    UF : 0, UT : 6,      CONFIG : 'N U T, 0, 0, 0',
    X =  237.679  mm,    Y =   97.904  mm,    Z =   677.007  mm,
    W =  -181.004 deg,    P =   0.018 deg,    R =   -1.000 deg
};
P[413]{
   GP1:
    UF : 0, UT : 6,      CONFIG : 'N U T, 0, 0, 0',
    X =  239.805  mm,    Y =   100.038  mm,    Z =   678.567  mm,
    W =  -180.980 deg,    P =   0.017 deg,    R =   -1.000 deg
};
P[414]{
   GP1:
    UF : 0, UT : 6,      CONFIG : 'N U T, 0, 0, 0',
    X =  237.603  mm,    Y =   102.637  mm,    Z =   678.250  mm,
    W =  -180.939 deg,    P =   0.016 deg,    R =   -1.000 deg
};
P[415]{
   GP1:
    UF : 0, UT : 6,      CONFIG : 'N U T, 0, 0, 0',
    X =  237.914  mm,    Y =   109.032  mm,    Z =   679.196  mm,
    W =  -180.916 deg,    P =   0.016 deg,    R =   -1.000 deg
};
P[416]{
   GP1:
    UF : 0, UT : 6,      CONFIG : 'N U T, 0, 0, 0',
    X =  238.466  mm,    Y =   114.556  mm,    Z =   679.491  mm,
    W =  -180.917 deg,    P =   0.016 deg,    R =   -1.000 deg
};
P[417]{
   GP1:
    UF : 0, UT : 6,      CONFIG : 'N U T, 0, 0, 0',
    X =  237.988  mm,    Y =   117.959  mm,    Z =   679.696  mm,
    W =  -180.951 deg,    P =   0.017 deg,    R =   -1.000 deg
};
P[418]{
   GP1:
    UF : 0, UT : 6,      CONFIG : 'N U T, 0, 0, 0',
    X =  237.933  mm,    Y =   124.350  mm,    Z =   679.696  mm,
    W =  -180.999 deg,    P =   0.017 deg,    R =   -1.000 deg
};
P[419]{
   GP1:
    UF : 0, UT : 6,      CONFIG : 'N U T, 0, 0, 0',
    X =  238.236  mm,    Y =   206.397  mm,    Z =   679.696  mm,
    W =  -180.000 deg,    P =   0.000 deg,    R =   0.000 deg
};
P[420]{
   GP1:
    UF : 0, UT : 6,      CONFIG : 'N U T, 0, 0, 0',
    X =  201.883  mm,    Y =   206.397  mm,    Z =   677.551  mm,
    W =  -180.000 deg,    P =   0.000 deg,    R =   0.000 deg
};
P[421]{
   GP1:
    UF : 0, UT : 6,      CONFIG : 'N U T, 0, 0, 0',
    X =  202.738  mm,    Y =   124.967  mm,    Z =   677.551  mm,
    W =  -181.191 deg,    P =   0.021 deg,    R =   -1.000 deg
};
P[422]{
   GP1:
    UF : 0, UT : 6,      CONFIG : 'N U T, 0, 0, 0',
    X =  202.486  mm,    Y =   119.434  mm,    Z =   677.551  mm,
    W =  -181.103 deg,    P =   0.019 deg,    R =   -1.000 deg
};
P[423]{
   GP1:
    UF : 0, UT : 6,      CONFIG : 'N U T, 0, 0, 0',
    X =  203.228  mm,    Y =   114.890  mm,    Z =   677.970  mm,
    W =  -180.965 deg,    P =   0.017 deg,    R =   -1.000 deg
};
P[424]{
   GP1:
    UF : 0, UT : 6,      CONFIG : 'N U T, 0, 0, 0',
    X =  202.797  mm,    Y =   108.893  mm,    Z =   678.745  mm,
    W =  -180.839 deg,    P =   0.015 deg,    R =   -1.000 deg
};
P[425]{
   GP1:
    UF : 0, UT : 6,      CONFIG : 'N U T, 0, 0, 0',
    X =  202.869  mm,    Y =   103.650  mm,    Z =   678.789  mm,
    W =  -180.846 deg,    P =   0.015 deg,    R =   -1.000 deg
};
P[426]{
   GP1:
    UF : 0, UT : 6,      CONFIG : 'N U T, 0, 0, 0',
    X =  202.572  mm,    Y =   100.291  mm,    Z =   678.701  mm,
    W =  -180.857 deg,    P =   0.015 deg,    R =   -1.000 deg
};
P[427]{
   GP1:
    UF : 0, UT : 6,      CONFIG : 'N U T, 0, 0, 0',
    X =  202.760  mm,    Y =   96.899  mm,    Z =   677.464  mm,
    W =  -180.877 deg,    P =   0.015 deg,    R =   -1.000 deg
};
P[428]{
   GP1:
    UF : 0, UT : 6,      CONFIG : 'N U T, 0, 0, 0',
    X =  203.006  mm,    Y =   91.575  mm,    Z =   677.087  mm,
    W =  -180.968 deg,    P =   0.017 deg,    R =   -1.000 deg
};
P[429]{
   GP1:
    UF : 0, UT : 6,      CONFIG : 'N U T, 0, 0, 0',
    X =  202.936  mm,    Y =   85.805  mm,    Z =   677.228  mm,
    W =  -181.086 deg,    P =   0.019 deg,    R =   -1.000 deg
};
P[430]{
   GP1:
    UF : 0, UT : 6,      CONFIG : 'N U T, 0, 0, 0',
    X =  202.752  mm,    Y =   80.302  mm,    Z =   677.133  mm,
    W =  -181.183 deg,    P =   0.021 deg,    R =   -1.000 deg
};
P[431]{
   GP1:
    UF : 0, UT : 6,      CONFIG : 'N U T, 0, 0, 0',
    X =  203.266  mm,    Y =   74.595  mm,    Z =   677.308  mm,
    W =  -181.243 deg,    P =   0.022 deg,    R =   -1.000 deg
};
P[432]{
   GP1:
    UF : 0, UT : 6,      CONFIG : 'N U T, 0, 0, 0',
    X =  202.857  mm,    Y =   69.136  mm,    Z =   677.567  mm,
    W =  -181.285 deg,    P =   0.022 deg,    R =   -1.000 deg
};
P[433]{
   GP1:
    UF : 0, UT : 6,      CONFIG : 'N U T, 0, 0, 0',
    X =  202.244  mm,    Y =   64.466  mm,    Z =   677.604  mm,
    W =  -181.312 deg,    P =   0.023 deg,    R =   -1.000 deg
};
P[434]{
   GP1:
    UF : 0, UT : 6,      CONFIG : 'N U T, 0, 0, 0',
    X =  202.914  mm,    Y =   58.122  mm,    Z =   677.421  mm,
    W =  -181.367 deg,    P =   0.024 deg,    R =   -1.000 deg
};
P[435]{
   GP1:
    UF : 0, UT : 6,      CONFIG : 'N U T, 0, 0, 0',
    X =  203.053  mm,    Y =   53.855  mm,    Z =   677.512  mm,
    W =  -181.395 deg,    P =   0.024 deg,    R =   -1.000 deg
};
P[436]{
   GP1:
    UF : 0, UT : 6,      CONFIG : 'N U T, 0, 0, 0',
    X =  202.843  mm,    Y =   46.563  mm,    Z =   675.931  mm,
    W =  -181.419 deg,    P =   0.025 deg,    R =   -1.000 deg
};
P[437]{
   GP1:
    UF : 0, UT : 6,      CONFIG : 'N U T, 0, 0, 0',
    X =  203.318  mm,    Y =   42.100  mm,    Z =   674.942  mm,
    W =  -181.434 deg,    P =   0.025 deg,    R =   -1.000 deg
};
P[438]{
   GP1:
    UF : 0, UT : 6,      CONFIG : 'N U T, 0, 0, 0',
    X =  202.881  mm,    Y =   39.256  mm,    Z =   674.563  mm,
    W =  -181.438 deg,    P =   0.025 deg,    R =   -1.000 deg
};
P[439]{
   GP1:
    UF : 0, UT : 6,      CONFIG : 'N U T, 0, 0, 0',
    X =  203.131  mm,    Y =   34.198  mm,    Z =   674.988  mm,
    W =  -181.441 deg,    P =   0.025 deg,    R =   -1.000 deg
};
P[440]{
   GP1:
    UF : 0, UT : 6,      CONFIG : 'N U T, 0, 0, 0',
    X =  202.832  mm,    Y =   28.738  mm,    Z =   675.954  mm,
    W =  -181.416 deg,    P =   0.025 deg,    R =   -1.000 deg
};
P[441]{
   GP1:
    UF : 0, UT : 6,      CONFIG : 'N U T, 0, 0, 0',
    X =  202.744  mm,    Y =   23.472  mm,    Z =   676.873  mm,
    W =  -181.376 deg,    P =   0.024 deg,    R =   -1.000 deg
};
P[442]{
   GP1:
    UF : 0, UT : 6,      CONFIG : 'N U T, 0, 0, 0',
    X =  202.866  mm,    Y =   17.338  mm,    Z =   677.956  mm,
    W =  -181.263 deg,    P =   0.022 deg,    R =   -1.000 deg
};
P[443]{
   GP1:
    UF : 0, UT : 6,      CONFIG : 'N U T, 0, 0, 0',
    X =  203.265  mm,    Y =   12.113  mm,    Z =   677.623  mm,
    W =  -181.138 deg,    P =   0.020 deg,    R =   -1.000 deg
};
P[444]{
   GP1:
    UF : 0, UT : 6,      CONFIG : 'N U T, 0, 0, 0',
    X =  202.579  mm,    Y =   6.550  mm,    Z =   676.710  mm,
    W =  -180.997 deg,    P =   0.017 deg,    R =   -1.000 deg
};
P[445]{
   GP1:
    UF : 0, UT : 6,      CONFIG : 'N U T, 0, 0, 0',
    X =  202.981  mm,    Y =   2.035  mm,    Z =   675.441  mm,
    W =  -180.903 deg,    P =   0.016 deg,    R =   -1.000 deg
};
P[446]{
   GP1:
    UF : 0, UT : 6,      CONFIG : 'N U T, 0, 0, 0',
    X =  201.883  mm,    Y =   -0.623  mm,    Z =   676.010  mm,
    W =  -180.856 deg,    P =   0.015 deg,    R =   -1.000 deg
};
P[447]{
   GP1:
    UF : 0, UT : 6,      CONFIG : 'N U T, 0, 0, 0',
    X =  202.866  mm,    Y =   -4.118  mm,    Z =   675.410  mm,
    W =  -180.726 deg,    P =   0.013 deg,    R =   -1.000 deg
};
P[448]{
   GP1:
    UF : 0, UT : 6,      CONFIG : 'N U T, 0, 0, 0',
    X =  202.877  mm,    Y =   -10.672  mm,    Z =   675.669  mm,
    W =  -180.524 deg,    P =   0.009 deg,    R =   -1.000 deg
};
P[449]{
   GP1:
    UF : 0, UT : 6,      CONFIG : 'N U T, 0, 0, 0',
    X =  202.997  mm,    Y =   -15.857  mm,    Z =   675.460  mm,
    W =  -180.390 deg,    P =   0.007 deg,    R =   -1.000 deg
};
P[450]{
   GP1:
    UF : 0, UT : 6,      CONFIG : 'N U T, 0, 0, 0',
    X =  202.823  mm,    Y =   -21.947  mm,    Z =   675.573  mm,
    W =  -180.109 deg,    P =   0.002 deg,    R =   -0.999 deg
};
P[451]{
   GP1:
    UF : 0, UT : 6,      CONFIG : 'N U T, 0, 0, 0',
    X =  203.057  mm,    Y =   -65.498  mm,    Z =   674.286  mm,
    W =  -179.305 deg,    P =   -0.012 deg,    R =   -0.996 deg
};
P[452]{
   GP1:
    UF : 0, UT : 6,      CONFIG : 'N U T, 0, 0, 0',
    X =  202.976  mm,    Y =   -71.266  mm,    Z =   674.286  mm,
    W =  -179.578 deg,    P =   -0.007 deg,    R =   -0.995 deg
};
P[453]{
   GP1:
    UF : 0, UT : 6,      CONFIG : 'N U T, 0, 0, 0',
    X =  201.883  mm,    Y =   -206.397  mm,    Z =   674.286  mm,
    W =  -180.000 deg,    P =   0.000 deg,    R =   0.000 deg
};
P[454]{
   GP1:
    UF : 0, UT : 6,      CONFIG : 'N U T, 0, 0, 0',
    X =  420.000  mm,    Y =   0.000  mm,    Z =   773.173  mm,
    W =  -180.000 deg,    P =   0.000 deg,    R =   0.000 deg
};
/END
